{attribute addProperty BoxType "EL4102--0000"}
{attribute addProperty Id "ChannelAT %Q*ARRAY[0..1] OF Channel_969D8B6C3240WcStateAT %I*WcState_28A8677510.1250InfoDataAT %I*InfoData_BC63D37F80100"}
{attribute addProperty CRC "1827809340"}
{attribute addProperty SizeInBites "113"}
{attribute addProperty SizeInBytes "14.125"}
TYPE EL4102_6AE7330D :
STRUCT
	{attribute addProperty Name "Channel"}
	Channel : ARRAY[0..1] OF Channel_969D8B6C;
	{attribute addProperty Name "WcState"}
	WcState : WcState_28A86775;
	{attribute addProperty Name "InfoData"}
	InfoData : InfoData_BC63D37F;
END_STRUCT
END_TYPE

(* stored: Version 1.2.0.0, ProductVersion 3.1.4024.9
   DUT EL4102_6AE7330D: Id {17a3b031-8743-4090-8f31-04592de450ff} *)
